# EPICS substitutions: icefrdgeSup/icefrdge_error_setter.substitutions
file $(UTILITIES)/db/error_setter.template {
    pattern {P, STREAM_PV, PV_NAME}

    {"\$(P)", "VTI:TEMP1", "VTI:TEMP2"}
    {"\$(P)", "VTI:TEMP1", "VTI:TEMP3"}
    {"\$(P)", "VTI:TEMP1", "VTI:TEMP4"}

    {"\$(P)", "LS:MC:P", "LS:MC:I"}
    {"\$(P)", "LS:MC:P", "LS:MC:D"}

    {"\$(P)", "MIMIC:PRESSURE1", "MIMIC:PRESSURE2"}
    {"\$(P)", "MIMIC:PRESSURE1", "MIMIC:PRESSURE3"}
    {"\$(P)", "MIMIC:PRESSURE1", "MIMIC:PRESSURE4"}

    {"\$(P)", "MC:TEMP", "MC:USER"}
}
